	sErrorDescription1 := ' Faulty wiring (Mode sel. swit.  The state of doubled wiring is not matching (Mode sel. switch).';				
	sErrorDescription2 := 'Please check the wiring (Mode sel. switch)';				
					
0047:					
					
	sErrorDescription1 := ' OCL detect.  OCL detect.';				
	sErrorDescription2 := 'Please check the line (O/P Emergency Stop)';				
					
0048:					
					
	sErrorDescription1 := ' Faulty line (Mode Selector SW.  The state of doubled line is not matching (Mode Selector switch).';				
	sErrorDescription2 := 'Please check the line (Mode Selector switch)';				
					
0049:					
					
	sErrorDescription1 := ' Faulty Line (T/B Enable Switc.  The state of doubled line is not matching (T/B Enable Switch).';				
	sErrorDescription2 := 'Please check the line (T/B Enable Switch)';				
					
0050:					
					
	sErrorDescription1 := 'EMG signal is input. (externa.  EMG signal is input. (external).';				
	sErrorDescription2 := 'Check the external emergency stop';				
					
0051:					
					
	sErrorDescription1 := 'EMG line is faulty.(external).  EMG line is faulty.(external).';				
	sErrorDescription2 := 'Check the external emergency stop';				
					
0052:					
					
	sErrorDescription1 := ' EMG signal is input.(Add.Axis.  EMG signal is input.(Add.Axis1).';				
	sErrorDescription2 := 'Check the emergency stop of Additional Axis card';				
					
0053:					
					
	sErrorDescription1 := 'EMG signal is input.(Add.Axis.  EMG signal is input.(Add.Axis).';				
	sErrorDescription2 := 'Check the emergency stop of Additional Axis servo amp.';				
					
0054:					
					
	sErrorDescription1 := ' Faulty wiring (External EMG p.  The state of doubled wiring is not matching (External EMG).';				
	sErrorDescription2 := 'Please check the wiring (External Emergency Stop)';				
					
0060:					
					
	sErrorDescription1 := 'EMG signal is input. (O.Panel.  EMG signal is input. (O.Panel).';				
	sErrorDescription2 := 'Check the O.Panel emergency stop';				
					
0061:					
					
	sErrorDescription1 := 'EMG line is faulty.(0.Panel).  EMG line is faulty.(0.Panel).';				
	sErrorDescription2 := 'Check the O.Panel emergency stop';				
					
0070:					
					
	sErrorDescription1 := 'EMG signal is input. (T.Box).  EMG signal is input. (T.Box).';				
	sErrorDescription2 := 'Check the T.Box emergency stop';				
					
0071:					
					
	sErrorDescription1 := 'EMG line is faulty.(T.Box).  EMG line is faulty.(T.Box).';				
	sErrorDescription2 := 'Check the T.Box emergency stop';				
					
0072:					
					
	sErrorDescription1 := 'EMG cancel operation is fault.  TB cancel switch operation was incorrect.';				
	sErrorDescription2 := 'Check the T/B cancel switch operation';				
					
0073:					
					
	sErrorDescription1 := 'EMG cancel line is faulty.(T..  EMG cancel line is faulty.(T.Box).';				
	sErrorDescription2 := 'Check the EMG cancel line';				
					
0074:					
					
	sErrorDescription1 := 'Faulty line (T/B Enable/Disab.  The state of doubled line is not matching (T/B Enable/Disable).';				
	sErrorDescription2 := 'Please check the line (T/B Enable/Disable)';				
					
0075:					
					
	sErrorDescription1 := 'TB communication error.  Communication between the RC and TB was cut off.';				
	sErrorDescription2 := 'Check TB communication line';				
					
0076:					
					
	sErrorDescription1 := 'TB connection error.  Cannot detect TB connection.';				
	sErrorDescription2 := 'If this error recurs, please contact us';				
					
0077:					
					
	sErrorDescription1 := ' Electric double layer overvol.  A power supply of a substrate in the robot is broken.';				
	sErrorDescription2 := 'Turn the power OFF and contact your service provider';				
					
0079:					
					
	sErrorDescription1 := ' Contactor of converter unit e.  Contactor of converter unit is closed.';				
	sErrorDescription2 := 'Confirm status of contactor of converter unit';				
					
0080:					
					
	sErrorDescription1 := ' Fuse of brake line is blown.  Fuse of brake line is blown.';				
	sErrorDescription2 := 'Change fuse';				
					
0081:					
					
	sErrorDescription1 := ' Fuse is blown.(motor hand I/F.  Fuse is blown.(motor hand I/F).';				
	sErrorDescription2 := 'Change fuse';				
					
0082:					
					
	sErrorDescription1 := 'Fuse is broken (air hand I/F).  Fuse is blown.(air hand I/F).';				
	sErrorDescription2 := 'Change fuse';				
					
0083:					
					
	sErrorDescription1 := 'Fuse is broken(hand input pow.  Fuse is blown.(hand input power).';				
	sErrorDescription2 := 'Change fuse';				
					
0084:					
					
	sErrorDescription1 := 'Fuse is broken(O/P).  Fuse is blown.(O/P).';				
	sErrorDescription2 := 'Change fuse';				
					
0085:					
					
	sErrorDescription1 := ' Fuse is blown.(External EMG).  Open phase in the input power.';				
	sErrorDescription2 := 'Change fuse';				
					
0086:					
					
	sErrorDescription1 := 'Hand module overcurrent.  Hand module is broken.';				
	sErrorDescription2 := 'Change Hand module';				
					
0087:					
					
	sErrorDescription1 := 'Fuse is blown.(Brake).  Fuse is blown.(Brake).';				
	sErrorDescription2 := 'Change fuse';				
					
0088:					
					
	sErrorDescription1 := ' Fuse is blown.(Service I/F).  Fuse is blown.(Service I/F).';				
	sErrorDescription2 := 'Please confirm the input and output current of service I/F. ';				
					
0089:					
					
	sErrorDescription1 := ' Fuse of external battery is b.  Fuse of external battery is blown..';				
	sErrorDescription2 := 'Check that an outside power-supply voltage is 4.5V or less.';				
					
0090:					
					
	sErrorDescription1 := ' Fuse is blown..  Fuse is blown.';				
	sErrorDescription2 := 'Change fuse';				
					
0093:					
					
	sErrorDescription1 := ' Safety relay fuse is blown..  Safety relay fuse is blown..';				
	sErrorDescription2 := 'Change fuse.';				
					
0094:					
					
	sErrorDescription1 := ' The fuse in the T/B was blown.  The fuse in the T/B power supply line was blown..';				
	sErrorDescription2 := 'Please check the earth fault of the T/B cable.';				
					
0097:					
					
	sErrorDescription1 := ' Faulty status (MC).  The state of doubled signal is not matching (MC status).';				
	sErrorDescription2 := 'Turn the power OFF and ON once';				
					
0098:					
					
	sErrorDescription1 := ' Faulty status (SR).  The state of doubled signal is not matching (SR status).';				
	sErrorDescription2 := 'Turn the power OFF and ON once';				
					
0099:					
					
	sErrorDescription1 := ' S/W with an old version is in.  S/W with an old version is installed.';				
	sErrorDescription2 := 'Install the S/W with a correct version';				
					
0100:					
					
	sErrorDescription1 := 'Temperature in the Controlle .  FAN check or Filter at the bottom on Controller becomes old.';				
	sErrorDescription2 := 'Please exchange the filter to new filter or clean up the filter';				
					
0103:					
					
	sErrorDescription1 := ' Temp. in robot CPU is too hig.  Ambient temperature of robot CPU becomes high.';				
	sErrorDescription2 := 'Please lower ambient temperature to the specification range';				
					
0117:					
					
	sErrorDescription1 := ' Power supply error (brake).  The output of the power supply deviated from the specified range.';				
	sErrorDescription2 := 'Turn the power OFF and contact your service provider';				
					
0130:					
					
	sErrorDescription1 := 'System RemoteI/O down.  Communication line of System Remote I/O is illegal.';				
	sErrorDescription2 := 'Check the cable or power supply';				
					
0131:					
					
	sErrorDescription1 := ' Plural Ope-panel are installe.  One operation panel can be installed..';				
	sErrorDescription2 := 'Install only one operation panel.';				
					
0140:					
					
	sErrorDescription1 := 'Fuse is blown.(Safety unit).  Fuse is blown.(Safety unit).';				
	sErrorDescription2 := 'Change fuse';				
					
0141:					
					
	sErrorDescription1 := ' Wiring error of EMGIN connect.  Wiring error of EMGIN connector.';				
	sErrorDescription2 := 'Please confirm the wiring for EMGIN';				
					
0160:					
					
	sErrorDescription1 := 'Cannot use PIO I/F and Unit.  The I/O Channel number of PIO interface and PIO unit overlaps..';				
	sErrorDescription2 := 'Select either of Paralle I/O interface or Paralle I/O unit.';				
					
0162:					
					
	sErrorDescription1 := 'Cannot use PIO I/F and Unit.  The I/O Channel number of PIO interface and PIO unit overlaps..';				
	sErrorDescription2 := 'Select either of Paralle I/O interface or Paralle I/O unit.';				
					
0163:					
					
	sErrorDescription1 := 'Cannot use PIO I/F and Unit.  The I/O Channel number of PIO interface and PIO unit overlaps..';				
	sErrorDescription2 := 'Select either of Paralle I/O interface or Paralle I/O unit.';				
					
0170:					
					
	sErrorDescription1 := 'Parallel I/O interface H/W er.  The card might be broken..';				
	sErrorDescription2 := 'Please exchange the Parallel I/O interface card.';				
					
0172:					
					
	sErrorDescription1 := 'Parallel I/O interface H/W er.  The card might be broken..';				
	sErrorDescription2 := 'Please exchange the Parallel I/O interface card.';				
					
0173:					
					
	sErrorDescription1 := 'Parallel I/O interface H/W er.  The card might be broken..';				
	sErrorDescription2 := 'Please exchange the Parallel I/O interface card.';				
					
0180:					
					
	sErrorDescription1 := 'Fuse is blown.(PIO) （Slot 1-F.  Fuse is blown.(Paralle I/O interface).';				
	sErrorDescription2 := 'Change fuse (Paralle I/O interface)';				
					
0182:					
					
	sErrorDescription1 := 'Fuse is blown.(PIO) （Slot 2-F.  Fuse is blown.(Paralle I/O interface).';				
	sErrorDescription2 := 'Change fuse (Paralle I/O interface)';				
					
0183:					
					
	sErrorDescription1 := 'Fuse is blown.(PIO) （Slot 3-F.  Fuse is blown.(Paralle I/O interface).';				
	sErrorDescription2 := 'Change fuse (Paralle I/O interface)';				
					
0210:					
					
	sErrorDescription1 := ' Power supply error.  The output of the power supply deviated from the specified range.';				
	sErrorDescription2 := 'Turn the power OFF and ON once';				
					
0211:					
					
	sErrorDescription1 := ' Power supply error.  The output of the power supply deviated from the specified range.';				
	sErrorDescription2 := 'Turn the power OFF and ON once';				
					
0212:					
					
	sErrorDescription1 := ' Power supply error.  The output of the power supply deviated from the specified range.';				
	sErrorDescription2 := 'Turn the power OFF and ON once';				
					
0213:					
					
	sErrorDescription1 := ' Power supply error.  The output of the power supply deviated from the specified range.';				
	sErrorDescription2 := 'Turn the power OFF and ON once';				
					
0220:					
					
	sErrorDescription1 := ' Memory error (Main CPU).  Memory error was detected (Main CPU).';				
	sErrorDescription2 := 'Turn the power OFF and ON once';				
					
0230:					
					
	sErrorDescription1 := ' Safety parameter error.  Detect errors in safety parameter value.';				
	sErrorDescription2 := 'Please check the safety parameter setting';				
					
0231:					
					
	sErrorDescription1 := ' Parameter CRC error.  Detect CRC errors in safety parameter.';				
	sErrorDescription2 := 'Please check the safety parameters settings and write parameters';				
					
0241:					
					
	sErrorDescription1 := ' Fault in Safety Communication.  Detect a fault in safety communication.';				
	sErrorDescription2 := 'Turn the power OFF and ON once';				
					
0242:					
					
	sErrorDescription1 := ' Fault in Safety Data.  Detect a fault in safety data.';				
	sErrorDescription2 := 'Turn the power OFF and ON once';				
					
0243:					
					
	sErrorDescription1 := ' Safety function unavailable.  The Safety Function is not supported by this robot.';				
	sErrorDescription2 := 'Disable the safety function';				
					
0260:					
					
	sErrorDescription1 := ' EMG circuit diagnosis error.  Voltage diagnosis error.';				
	sErrorDescription2 := 'Turn the power OFF and ON once';				
					
0270:					
					
	sErrorDescription1 := ' Voltage diagnosis error.  Voltage diagnosis error.';				
	sErrorDescription2 := 'Turn the power OFF and ON once';				
					
0280:					
					
	sErrorDescription1 := ' STO circuit diagnosis error.  STO citcuit error.';				
	sErrorDescription2 := 'Turn the power OFF and ON once';				
					
0290:					
					
	sErrorDescription1 := ' PLD control error.  PLD control error.';				
	sErrorDescription2 := 'Turn the power OFF and ON once';				
					
0300:					
					
	sErrorDescription1 := ' CR800 test H-Error.  General-purpose H-Error for the function test of CR800.';				
	sErrorDescription2 := 'Check the embedded message';				
					
0310:					
					
	sErrorDescription1 := ' Mecha board access error.  Failed in access to a Mecha board.';				
	sErrorDescription2 := 'Please confirm the connection with Mecha board';				
					
0311:					
					
	sErrorDescription1 := ' RemoteI/O unit config error.  The multiple RemoteI/O units which do not support are connected.';				
	sErrorDescription2 := 'Please confirm the constitution of RemoteI/O unit';				
					
0315:					
					
	sErrorDescription1 := ' Can not access the D-device are.  This area cannot be used in duplicate.';				
	sErrorDescription2 := 'Please change the D-device start number in parameter DDEVVLn';				
					
0316:					
					
	sErrorDescription1 := ' The D-device area is out of r.  An area corresponding to the variable type can not be allocated.';				
	sErrorDescription2 := 'Please change the D-device start number in parameter DDEVVLn';				
					
0317:					
					
	sErrorDescription1 := ' The D-device variable duplica.  Cannot be doubly allotted to one variable.';				
	sErrorDescription2 := 'Please change the variable name in parameter DDEVVLn';				
					
0470:					
					
	sErrorDescription1 := ' Abnormality of DB(Add.Axis).  The addition axis dynamic brake is abnormal.';				
	sErrorDescription2 := 'Check the dynamic brake unit and the cable connection';				
					
0490:					
					
	sErrorDescription1 := 'Alarm of fan in the robot.  Fan in the robot might be out of order.';				
	sErrorDescription2 := 'Please exchange the fan in the robot';				
					
0491:					
					
	sErrorDescription1 := 'Alarm of fan1 in the robot.  Fan1 in the robot might be out of order.';				
	sErrorDescription2 := 'Please exchange the fan1 in the robot';				
					
0492:					
					
	sErrorDescription1 := 'Alarm of fan2 in the robot.  Fan2 in the robot might be out of order.';				
	sErrorDescription2 := 'Please exchange the fan2 in the robot';				
					
0493:					
					
	sErrorDescription1 := 'Alarm of fan3 in the robot.  Fan3 in the robot might be out of order.';				
	sErrorDescription2 := 'Please exchange the fan3 in the robot';				
					
0494:					
					
	sErrorDescription1 := 'Alarm of fan4 in the robot.  Fan4 in the robot might be out of order.';				
	sErrorDescription2 := 'Please exchange the fan4 in the robot';				
					
0495:					
					
	sErrorDescription1 := 'Alarm of fan5 in the robot.  Fan5 in the robot might be out of order.';				
	sErrorDescription2 := 'Please exchange the fan5 in the robot';				
					
0496:					
					
	sErrorDescription1 := 'Alarm of fan6 in the robot.  Fan6 in the robot might be out of order.';				
	sErrorDescription2 := 'Please exchange the fan6 in the robot';				
					
0497:					
					
	sErrorDescription1 := 'Alarm of fan7 in the robot.  Fan7 in the robot might be out of order.';				
	sErrorDescription2 := 'Please exchange the fan7 in the robot';				
					
0498:					
					
	sErrorDescription1 := 'Alarm of fan8 in the robot.  Fan8 in the robot might be out of order.';				
	sErrorDescription2 := 'Please exchange the fan8 in the robot';				
					
0500:					
					
	sErrorDescription1 := 'Servo axis setting error.  The setting of the axis number selection switch is illegal.';				
	sErrorDescription2 := 'Confirm the setting of the axis selection switch';				
					
0510:					
					
	sErrorDescription1 := 'The converter setting is ille.  The setting of the external emergency stop mode is illegal.';				
	sErrorDescription2 := 'Correctly set';				
					
0520:					
					
	sErrorDescription1 := 'Robot axis setting illegal.  The axis No is duplicated with another robot axis No.';				
	sErrorDescription2 := 'Correctly set';				
					
0530:					
					
	sErrorDescription1 := 'Servo sys. error (memory).  The servo amplifier memory ICs check sum is illegal.';				
	sErrorDescription2 := 'Turn the power OFF and ON once';				
					
0540:					
					
	sErrorDescription1 := 'Servo sys. error (over run).  The servo amp. / motion task S/W did not end within the specified time.';				
	sErrorDescription2 := 'Turn the power OFF and ON once';				
					
0550:					
					
	sErrorDescription1 := 'Servo sys. error (mag. pole p.  the magnetic pole position signal from encoderis illegal.';				
	sErrorDescription2 := 'Turn the power OFF and ON once';				
					
0560:					
					
	sErrorDescription1 := 'Servo sys. error (A/D）.  the magnetic pole position signal from encoderis illegal.';				
	sErrorDescription2 := 'Turn the power OFF and ON once';				
					
0570:					
					
	sErrorDescription1 := 'Encoder error (EEPROM).  the magnetic pole position signal from encoderis illegal.';				
	sErrorDescription2 := 'Turn the power OFF and ON once';				
					
0580:					
					
	sErrorDescription1 := 'Encoder error (LED).  The LED of encoder has deteriorated.';				
	sErrorDescription2 := 'Turn the power OFF and ON once';				
					
0590:					
					
	sErrorDescription1 := 'Encoder error (position data).  the per rotation position data is illegal.';				
	sErrorDescription2 := 'Turn the power OFF and ON once';				
					
0600:					
					
	sErrorDescription1 := 'Encoder no-signal detection1.  An error was detected in the operation input of the encoder.';				
	sErrorDescription2 := 'Turn the power OFF and ON once';				
					
0610:					
					
	sErrorDescription1 := 'Encoder no-signal detection2.  An error was detected in the operation input of the encoder.';				
	sErrorDescription2 := 'Turn the power OFF and ON once';				
					
0620:					
					
	sErrorDescription1 := 'Servo amplifier LSI error.  An error was detected in the operation of the servo AMP LSI.';				
	sErrorDescription2 := 'Turn the power OFF and ON once';				
					
0630:					
					
	sErrorDescription1 := 'Unused axis servo error.  A power module error occurred in an axis not used.';				
	sErrorDescription2 := 'Turn the power OFF and ON once';				
					
0640:					
					
	sErrorDescription1 := 'System error (ABS CPU).  Error in the CPU of the absolute position linear scale.';				
	sErrorDescription2 := 'Turn the power OFF and ON once';				
					
0650:					
					
	sErrorDescription1 := 'Absolute position error.  Error in the circuit of the absolute position linear scale.';				
	sErrorDescription2 := 'Turn the power OFF and ON once';				
					
0660:					
					
	sErrorDescription1 := 'Incremental position error.  Error in the incremental position detection circuit.';				
	sErrorDescription2 := 'Turn the power OFF and ON once';				
					
0670:					
					
	sErrorDescription1 := 'Encoder CPU error.  An error was detected in the CPU of the encoder.';				
	sErrorDescription2 := 'Turn the power OFF and ON once';				
					
0680:					
					
	sErrorDescription1 := 'Encoder LED error.  Deterioration of the encoder LED was detected.';				
	sErrorDescription2 := 'Turn the power OFF and ON once';				
					
0690:					
					
	sErrorDescription1 := ' regeneration circuit error.  A regenerative transistor or resistor error was detected.';				
	sErrorDescription2 := 'Turn the power OFF and ON once';				
					
0700:					
					
	sErrorDescription1 := 'P.S. external contactor fusin.  The external contactor turned ON even at READY OFF.';				
	sErrorDescription2 := 'Turn the power OFF and ON once';				
					
0710:					
					
	sErrorDescription1 := 'Power supply rush relay error.  The relay on servo cpu card did not turn ON.';				
	sErrorDescription2 := 'Turn the power OFF and ON once';				
					
0711:					
					
	sErrorDescription1 := 'Power supply relay error.  The discharge relay on converter card did not turn ON.';				
	sErrorDescription2 := 'Turn the power OFF and ON once';				
					
0712:					
					
	sErrorDescription1 := ' Converter fuse fusing.  Fuse of a converter fused for a ground fault or short circuit.';				
	sErrorDescription2 := 'Please exchange a fuse of a converter';				
					
0713:					
					
	sErrorDescription1 := ' Encoder power supply fuse tri.  Encoder power supply fuse tripped by ground fault, short circuit.';				
	sErrorDescription2 := 'Turn the power OFF, wait a while, and then turn ON again';				
					
0720:					
					
	sErrorDescription1 := 'Power supply watch dog.  The power supply S/W did not end within the specified time.';				
	sErrorDescription2 := 'Turn the power OFF and ON once';				
					
0730:					
					
	sErrorDescription1 := 'Power supply rush relay fusin.  The rush resistance short-circuit relay did not turn OFF.';				
	sErrorDescription2 := 'Turn the power OFF and ON once';				
					
0740:					
					
	sErrorDescription1 := 'Power supply main circuit err.  The main circuit capacitor was not charged correctly.';				
	sErrorDescription2 := 'Turn the power OFF and ON once';				
					
0742:					
					
	sErrorDescription1 := ' Power supply main circuit err.  A main circuit voltage has decreased because of Safety relay.';				
	sErrorDescription2 := 'Check for errors in the Safety relay';				
					
0743:					
					
	sErrorDescription1 := ' Power supply main circuit err.  A main circuit voltage has decreased because of contactor fail..';				
	sErrorDescription2 := 'Check for errors in the contactor.';				
					
0750:					
					
	sErrorDescription1 := 'Power supply memory error.  An error was detected in the power supply memory circuit.';				
	sErrorDescription2 := 'Turn the power OFF and ON once';				
					
0760:					
					
	sErrorDescription1 := 'Power supply error.  An error was detected in the data comm. with the power supply.';				
	sErrorDescription2 := 'Turn the power OFF and ON once';				
					
0770:					
					
	sErrorDescription1 := 'Power supply process error.  An error occurred in the process cycle of power supply.';				
	sErrorDescription2 := 'Turn the power OFF and ON once';				
					
0780:					
					
	sErrorDescription1 := 'Servo amplifier watch dog.  The Servo amplifier S/W did not end within the specified time.';				
	sErrorDescription2 := 'Turn the power OFF and ON once';				
					
0790:					
					
	sErrorDescription1 := 'Servo amplifier boad error.  An error was detected in the servo amplifier PCB.';				
	sErrorDescription2 := 'Turn the power OFF and ON once';				
					
0800:					
					
	sErrorDescription1 := 'Servo amplifier clock error.  An error was detected in the servo amplifier clock.';				
	sErrorDescription2 := 'Turn the power OFF and ON once';				
					
0810:					
					
	sErrorDescription1 := 'Power supply undervoltage.  Insufficient bus voltage was detected in main circuit.';				
	sErrorDescription2 := 'Check the power supply connection and power supply state';				
					
0820:					
					
	sErrorDescription1 := 'Motor ground fault.  A motor cable ground fault was detected.';				
	sErrorDescription2 := 'Check the motor cables connection and conductivity';				
					
0830:					
					
	sErrorDescription1 := 'Servo amplifier overvoltage.  The main circuit bus voltage exceeded the tolerable value.';				
	sErrorDescription2 := 'Check the power voltage and regenerative resistance value';				
					
0840:					
					
	sErrorDescription1 := 'Instantaneous power failure(S.  The power was OFF for 50msec or more.';				
	sErrorDescription2 := 'Check the power supply connection and power supply state';				
					
0850:					
					
	sErrorDescription1 := 'Power supply voltage incorrec.  Open phase in the input power, or the voltage is outof range.';				
	sErrorDescription2 := 'Check the power supply connection and power supply state';				
					
0860:					
					
	sErrorDescription1 := 'Power supply overvoltage.  The main circuit bus voltage exceeded the tolerable value.';				
	sErrorDescription2 := 'Check the power supply connection and power supply state';				
					
0870:					
					
	sErrorDescription1 := 'Power module overheat (Fan St.  A cooling fan stopped, and overheat occurred.';				
	sErrorDescription2 := 'Check the rotation of fan, and the connector connected to a fan';				
					
0880:					
					
	sErrorDescription1 := 'Power module overheat.  Overheating of the power module (IPM) was detected.';				
	sErrorDescription2 := 'Turn the power OFF, wait a while, and then turn ON again';				
					
0890:					
					
	sErrorDescription1 := 'Servo amplifier motor overhea.  The motor or detectors thermal protector activated.';				
	sErrorDescription2 := 'Turn the power OFF, wait a while, and then turn ON again';				
					
0900:					
					
	sErrorDescription1 := 'Absolute position overspeed.  The absolute position linear scale moved 45mm/s or more.';				
	sErrorDescription2 := 'Turn the power OFF and ON once';				
					
0910:					
					
	sErrorDescription1 := 'Servo amplifier overspeed.  The motor speed rose to 1.2 times the rating.';				
	sErrorDescription2 := 'Turn the power OFF and ON once';				
					
0920:					
					
	sErrorDescription1 := 'Power module overcurrent.  An overcurrent was detected in the  power supply IPM.';				
	sErrorDescription2 := 'Check the motor cables connection and conductivity';				
					
0930:					
					
	sErrorDescription1 := 'Motor overcurrent.  An excessive current flowed to the motor.';				
	sErrorDescription2 := 'Turn the power OFF and ON once';				
					
0940:					
					
	sErrorDescription1 := 'Overload 1.  Run in the overload range set with SVOLL and SVOLT.';				
	sErrorDescription2 := 'Check the load weight and the robot for collisions, etc';				
					
0950:					
					
	sErrorDescription1 := 'Overload 2.  95% or more of max current command continued for 1 sec. or more.';				
	sErrorDescription2 := 'Check the load weight and the robot for collisions, etc';				
					
0960:					
					
	sErrorDescription1 := 'Excessive error 1.  The position error exceeded at servo ON.';				
	sErrorDescription2 := 'Check the load weight and press, etc';				
					
0970:					
					
	sErrorDescription1 := 'Excessive error 2.  The position error exceeded at servo OFF.';				
	sErrorDescription2 := 'Check the moving robot arm by something power';				
					
0980:					
					
	sErrorDescription1 := 'Excessive error 3.  Abnormal motor power line connection.';				
	sErrorDescription2 := 'Check the connection of motor power line';				
					
0990:					
					
	sErrorDescription1 := 'Collision detection 0.  A collision detection method 1 error was detected during the G0.';				
	sErrorDescription2 := 'Release the collision state';				
					
1000:					
					
	sErrorDescription1 := 'Collision detection 1.  A collision detection method 1 error was detected during the G1.';				
	sErrorDescription2 := 'Release the collision state';				
					
1010:					
					
	sErrorDescription1 := 'Collision detection.  Robot collided with something, or COLLVL is too low.';				
	sErrorDescription2 := 'Removal of the factor of a collision, or improve COLLVL';				
					
1020:					
					
	sErrorDescription1 := 'Servo AMP over-regeneration.  Overheating of the regenerative resistor was detected.';				
	sErrorDescription2 := 'Check the regeneration capacity and parameter SVPTYPE';				
					
1030:					
					
	sErrorDescription1 := 'Power supply over-regeneratio.  The power supplys regeneration capacity limit was exceeded.';				
	sErrorDescription2 := 'Wait at least 15min in the power ON state, and then turn OFF';				
					
1040:					
					
	sErrorDescription1 := 'Encoder init communication er.  Initial communication with the encoder was not possible.';				
	sErrorDescription2 := 'Check the encoder cable connection';				
					
1050:					
					
	sErrorDescription1 := ' Encoder init communication er.  Initial communication with the encoder was not possible.';				
	sErrorDescription2 := 'Check the encoder cable connection';				
					
1060:					
					
	sErrorDescription1 := ' Encoder communication error.  Communication between the encoder and detector was cut off.';				
	sErrorDescription2 := 'Check the encoder cable connection';				
					
1070:					
					
	sErrorDescription1 := 'Encoder communication error.  Communication between the encoder and detector was cut off.';				
	sErrorDescription2 := 'Check the encoder cable connection';				
					
1080:					
					
	sErrorDescription1 := 'Servo AMP communication error.  Communication from the RC was cut off.';				
	sErrorDescription2 := 'Check the communication cable connection and conductivity';				
					
1090:					
					
	sErrorDescription1 := 'Servo AMP initialization erro.  Initialization of the servo amplifier failed.';				
	sErrorDescription2 := 'Check the servo axis settings (parameters, rotary switches)';				
					
1100:					
					
	sErrorDescription1 := 'Servo com. receive error.  Abnormality occurred in data reception from a servo amplifier.';				
	sErrorDescription2 := 'Check the communication cable connection and conductivity';				
					
1110:					
					
	sErrorDescription1 := 'Servo com. receive error.  Abnormality occurred in data reception from a servo amplifier.';				
	sErrorDescription2 := 'Check the communication cable connection and conductivity';				
					
1120:					
					
	sErrorDescription1 := 'Encoder ABS position data los.  The absolute position data in the detector was lost.';				
	sErrorDescription2 := 'Check the battery voltage and detector cable';				
					
1130:					
					
	sErrorDescription1 := 'Encoder per rotation data err.  An error was detected in the encoders per rotation data.';				
	sErrorDescription2 := 'Check the repeatability and ambient environment';				
					
1140:					
					
	sErrorDescription1 := 'SRV-AMP Comm. data error (CRC.  A CRC error was detected in the data from the RC.';				
	sErrorDescription2 := 'Check the communication cable connection and conductivity';				
					
1150:					
					
	sErrorDescription1 := 'Large command position.  The command position from the RC is abnormally large.';				
	sErrorDescription2 := 'Check the communication cable connection and conductivity';				
					
1160:					
					
	sErrorDescription1 := 'SRV-AMP Comm. error (frame).  An error was detected in the communication frame from the RC.';				
	sErrorDescription2 := 'Check the communication cable connection and conductivity';				
					
1170:					
					
	sErrorDescription1 := 'SRV-AMP Comm. error (info).  Error in the communication information from the RC.';				
	sErrorDescription2 := 'Check the communication cable connection and conductivity';				
					
1180:					
					
	sErrorDescription1 := 'Servo amplifier feedback erro.  A pulse was skipped in the detector feedback signal.';				
	sErrorDescription2 := 'Check the encoder cable connection and conductivity';				
					
1190:					
					
	sErrorDescription1 := 'Servo amplifier feedback erro.  A deviation occurred in the motor end and machine end positions.';				
	sErrorDescription2 := 'Check the encoder';				
					
1200:					
					
	sErrorDescription1 := 'SRV-AMP Comm. data error (CRC.  CRC error in the communication data from the servo amplifier.';				
	sErrorDescription2 := 'Check the communication cable connection and conductivity';				
					
1210:					
					
	sErrorDescription1 := 'SRV-AMP Comm. data error (ID).  Data ID error in the communication data from the servo AMP.';				
	sErrorDescription2 := 'Check the communication cable connection and conductivity';				
					
1220:					
					
	sErrorDescription1 := 'SRV-AMP Comm. data error(axis.  Axis No error in the communication data from the servo AMP.';				
	sErrorDescription2 := 'Check the communication cable connection and conductivity';				
					
1230:					
					
	sErrorDescription1 := 'SRV-AMP Comm. data error(SubI.  Sub ID error in the communication data from the servo AMP.';				
	sErrorDescription2 := 'Check the communication cable connection and conductivity';				
					
1240:					
					
	sErrorDescription1 := 'SRV-AMP Comm. data error(fram.  No. of frames error in the communication data from servo AMP.';				
	sErrorDescription2 := 'Check the communication cable connection and conductivity';				
					
1250:					
					
	sErrorDescription1 := 'Servo amplifier parameter err.  An error was detected in the servo parameter.';				
	sErrorDescription2 := 'Change the servo parameter to an appropriate value';				
					
1360:					
					
	sErrorDescription1 := ' Absolute position counter err.  The counter of absolute position is illegal.';				
	sErrorDescription2 := 'Check the repeatability and ambient environment';				
					
1380:					
					
	sErrorDescription1 := ' Removing control axis (servo).  The axis removable command has been input from the controller.';				
	sErrorDescription2 := 'Reset the axis removable command';				
					
1390:					
					
	sErrorDescription1 := 'Emergency stop (Servo amplifi.  The emergency stop command has been input from the RC.';				
	sErrorDescription2 := 'Release the emergency stop state';				
					
1410:					
					
	sErrorDescription1 := 'Instantaneous power failure(S.  The power was momentarily interrupted.';				
	sErrorDescription2 := 'Check power spec., and wiring of power and external EMG. stop';				
					
1440:					
					
	sErrorDescription1 := 'System error (servo 1).  Trouble occurred in the current processing CPU.';				
	sErrorDescription2 := 'Turn the power OFF and ON';				
					
1450:					
					
	sErrorDescription1 := 'Instantaneous power interrupt.  The power was momentarily interrupted at the power supply.';				
	sErrorDescription2 := 'Check power spec., and wiring of power and external EMG. stop';				
					
1460:					
					
	sErrorDescription1 := 'Power supply overcurrent.  Overcurrent in the power module in the power supply.';				
	sErrorDescription2 := 'Check the AC power line, or change the power supply';				
					
1470:					
					
	sErrorDescription1 := 'Frequency error.  AC frequency is out of range.';				
	sErrorDescription2 := 'Check the AC power line frequency, or change the power supply';				
					
1480:					
					
	sErrorDescription1 := 'Power supply parameter error.  Illegal at the power supply parameter.';				
	sErrorDescription2 := 'Set the correct parameter';				
					
1490:					
					
	sErrorDescription1 := 'Power supply overheat.  Overheating of the power module or regenerative resistance.';				
	sErrorDescription2 := 'Check the fan on rear of power supply';				
					
1491:					
					
	sErrorDescription1 := ' Illegal converter thermal  se.  Overheating of  servo AMP converter..';				
	sErrorDescription2 := 'Turn the power OFF, wait a while, and then turn ON again.';				
					
1492:					
					
	sErrorDescription1 := ' Power supply converter overhe.  Overheating of the converter was detected.';				
	sErrorDescription2 := 'Turn the power OFF, wait a while, and then turn ON again';				
					
1493:					
					
	sErrorDescription1 := ' Rush resistance overheat.  Overheating of the rush resistance was detected.';				
	sErrorDescription2 := 'Turn the power OFF, wait a while, and then turn ON again';				
					
1494:					
					
	sErrorDescription1 := ' Discharge resistance overheat.  Overheating of the discharge resistance was detected.';				
	sErrorDescription2 := 'Turn the power OFF, wait a while, and then turn ON again';				
					
1500:					
					
	sErrorDescription1 := 'Motor combination error.  Illegal combination with additional servo amp and motor.';				
	sErrorDescription2 := 'Use additional servo amp with correctly combination';				
					
1510:					
					
	sErrorDescription1 := 'SRV-AMP USB comm. Error.  A communication error was detected between the servo amp and PC.';				
	sErrorDescription2 := 'Check the communication cable connection and conductivity';				
					
1530:					
					
	sErrorDescription1 := ' Encoder memory error.  .';				
	sErrorDescription2 := '';				
					
1540:					
					
	sErrorDescription1 := 'Communication error between u.  The transmission data between servo amplifier units is illegal.';				
	sErrorDescription2 := 'Check the communication cable connection and conductivity';				
					
1550:					
					
	sErrorDescription1 := 'Emergency stop is a breakdown.  The external emergency stop input is illegal.';				
	sErrorDescription2 := 'Turn the power OFF and ON once';				
					
1561:					
					
	sErrorDescription1 := 'Excessive error 4.  Axis moved during servo on process.';				
	sErrorDescription2 := 'It is necessary to change some parts when not improvement';				
					
1570:					
					
	sErrorDescription1 := 'Non-registered servo error.  A non-registered servo error occurred.';				
	sErrorDescription2 := 'If the warning cannot be reset, turn the power OFF and ON';				
					
1590:					
					
	sErrorDescription1 := ' System error (illegal EMG).  An non-registered emergency stop was input.';				
	sErrorDescription2 := '';				
					
1600:					
					
	sErrorDescription1 := 'System error (No robot setted.  None of the robots are set.';				
	sErrorDescription2 := 'Set the robots for at least one unit';				
					
1601:					
					
	sErrorDescription1 := ' Unmatched robot model.  Robot arm that connection is not correct.';				
	sErrorDescription2 := 'Please confirm the connected robot arm';				
					
1610:					
					
	sErrorDescription1 := 'System error (illegal MEMECH).  The setting parameter MEMECH is illegal.';				
	sErrorDescription2 := 'Set the correct MEMECH';				
					
1680:					
					
	sErrorDescription1 := 'Cannot servo ON (timeout).  The servo did not turn ON within the specified time.';				
	sErrorDescription2 := 'Check for errors in the servo amplifier';				
					
1681:					
					
	sErrorDescription1 := 'Unexpected servo OFF.  The servo turned OFF unexpectedly.';				
	sErrorDescription2 := 'Check for errors in the servo amplifier';				
					
1682:					
					
	sErrorDescription1 := ' Servo ON Timeout(Safety relay.  A main circuit voltage did not rise because of Safety relay.';				
	sErrorDescription2 := 'Check for errors in the Safety relay';				
					
1683:					
					
	sErrorDescription1 := ' Servo ON Timeout.(Contactor).  A main circuit voltage did not rise because of contactor welded..';				
	sErrorDescription2 := 'Check for errors in the contactor.';				
					
1790:					
					
	sErrorDescription1 := 'Illegal parameter (MEJAR).  The setting of parameter MEJAR is illegal.';				
	sErrorDescription2 := 'Correct the parameter MEJAR';				
					
1800:					
					
	sErrorDescription1 := 'Illegal parameter (MEMAR).  The setting of parameter MEMAR is illegal.';				
	sErrorDescription2 := 'Correct the parameter MEMAR';				
					
1810:					
					
	sErrorDescription1 := 'Illegal parameter (USERORG).  The setting of parameter USERORG is illegal.';				
	sErrorDescription2 := 'Correct the parameter USERORG';				
					
1861:					
					
	sErrorDescription1 := 'Illegal parameter (J1OFFSET).  The setting of parameter J1OFFSET is illegal.';				
	sErrorDescription2 := 'Correct the 2nd element of parameter J1OFFSET';				
					
1881:					
					
	sErrorDescription1 := 'Cooling fan stopped (add. axi.  Cooling fan of the add. axis amp. J1 might be out of order.';				
	sErrorDescription2 := 'Please exchange the cooling fan';				
					
1882:					
					
	sErrorDescription1 := 'Cooling fan stopped (add. axi.  Cooling fan of the add. axis amp. J2 might be out of order.';				
	sErrorDescription2 := 'Please exchange the cooling fan';				
					
1883:					
					
	sErrorDescription1 := 'Cooling fan stopped (add. axi.  Cooling fan of the add. axis amp. J3 might be out of order.';				
	sErrorDescription2 := 'Please exchange the cooling fan';				
					
1884:					
					
	sErrorDescription1 := 'Cooling fan stopped (add. axi.  Cooling fan of the add. axis amp. J4 might be out of order.';				
	sErrorDescription2 := 'Please exchange the cooling fan';				
					
1885:					
					
	sErrorDescription1 := 'Cooling fan stopped (add. axi.  Cooling fan of the add. axis amp. J5 might be out of order.';				
	sErrorDescription2 := 'Please exchange the cooling fan';				
					
1886:					
					
	sErrorDescription1 := 'Cooling fan stopped (add. axi.  Cooling fan of the add. axis amp. J6 might be out of order.';				
	sErrorDescription2 := 'Please exchange the cooling fan';				
					
1887:					
					
	sErrorDescription1 := 'Cooling fan stopped (add. axi.  Cooling fan of the add. axis amp. J7 might be out of order.';				
	sErrorDescription2 := 'Please exchange the cooling fan';				
					
1888:					
					
	sErrorDescription1 := 'Cooling fan stopped (add. axi.  Cooling fan of the add. axis amp. J8 might be out of order.';				
	sErrorDescription2 := 'Please exchange the cooling fan';				
					
1900:					
					
	sErrorDescription1 := 'Cooling fan stopped (pow. sup.  The power supply cooling fan stopped.';				
	sErrorDescription2 := 'Confirm the rotation of the power supply cooling fan';				
					
1950:					
					
	sErrorDescription1 := ' Additional axis AMP error.  Alarm of the additional axis servo amplifier was detected.';				
	sErrorDescription2 := 'Please refer to the manual of servo amplifier.';				
					
2031:					
					
	sErrorDescription1 := 'Illegal parameter(JOGTSJ,JOGJ.  Illegal parameter(JOGTSJ,JOGJSP).';				
	sErrorDescription2 := 'Set value under 5';				
					
2090:					
					
	sErrorDescription1 := 'In interference zone n.  Movement inside the user-defined area range was attempted.';				
	sErrorDescription2 := 'Adjust the position data';				
					
2111:					
					
	sErrorDescription1 := 'Free plane 1 overrun.  Movement outside the free plane 1 was attempted.';				
	sErrorDescription2 := 'Change the position data';				
					
2112:					
					
	sErrorDescription1 := 'Free plane 2 overrun.  Movement outside the free plane 2 was attempted.';				
	sErrorDescription2 := 'Change the position data';				
					
2113:					
					
	sErrorDescription1 := 'Free plane 3 overrun.  Movement outside the free plane 3 was attempted.';				
	sErrorDescription2 := 'Change the position data';				
					
2114:					
					
	sErrorDescription1 := 'Free plane 4 overrun.  Movement outside the free plane 4 was attempted.';				
	sErrorDescription2 := 'Change the position data';				
					
2115:					
					
	sErrorDescription1 := 'Free plane 5 overrun.  Movement outside the free plane 5 was attempted.';				
	sErrorDescription2 := 'Change the position data';				
					
2116:					
					
	sErrorDescription1 := 'Free plane 6 overrun.  Movement outside the free plane 6 was attempted.';				
	sErrorDescription2 := 'Change the position data';				
					
2117:					
					
	sErrorDescription1 := 'Free plane 7 overrun.  Movement outside the free plane 7 was attempted.';				
	sErrorDescription2 := 'Change the position data';				
					
2118:					
					
	sErrorDescription1 := 'Free plane 8 overrun.  Movement outside the free plane 8 was attempted.';				
	sErrorDescription2 := 'Change the position data';				
					
2119:					
					
	sErrorDescription1 := ' Free plane 9 overrun.  Movement outside the free plane 9 was attempted.';				
	sErrorDescription2 := 'Change the position data';				
					
2120:					
					
	sErrorDescription1 := ' Free plane 10 overrun.  Movement outside the free plane 10 was attempted.';				
	sErrorDescription2 := 'Change the position data';				
					
2121:					
					
	sErrorDescription1 := ' Free plane 11 overrun.  Movement outside the free plane 11 was attempted.';				
	sErrorDescription2 := 'Change the position data';				
					
2122:					
					
	sErrorDescription1 := ' Free plane 12 overrun.  Movement outside the free plane 12 was attempted.';				
	sErrorDescription2 := 'Change the position data';				
					
2123:					
					
	sErrorDescription1 := ' Free plane 13 overrun.  Movement outside the free plane 13 was attempted.';				
	sErrorDescription2 := 'Change the position data';				
					
2124:					
					
	sErrorDescription1 := ' Free plane 14 overrun.  Movement outside the free plane 14 was attempted.';				
	sErrorDescription2 := 'Change the position data';				
					
2125:					
					
	sErrorDescription1 := ' Free plane 15 overrun.  Movement outside the free plane 15 was attempted.';				
	sErrorDescription2 := 'Change the position data';				
					
2126:					
					
	sErrorDescription1 := ' Free plane 16 overrun.  Movement outside the free plane 16 was attempted.';				
	sErrorDescription2 := 'Change the position data';				
					
2129:					
					
	sErrorDescription1 := 'Free plane limit data illegal.  The free plane data setting value is illegal.';				
	sErrorDescription2 := 'Set the correct free plane setting data';				
					
2130:					
					
	sErrorDescription1 := 'Speed is excessive (command).  The axis speed limit was exceeded.';				
	sErrorDescription2 := 'Reduce the robot motion speed,insert an OVRD,ACCEL or SPD';				
					
2131:					
					
	sErrorDescription1 := 'J1 Speed is excessive (comman.  The axis J1 speed limit was exceeded.';				
	sErrorDescription2 := 'Reduce the robot motion speed,insert an OVRD,ACCEL or SPD';				
					
2132:					
					
	sErrorDescription1 := 'J2 Speed is excessive (comman.  The axis J2 speed limit was exceeded.';				
	sErrorDescription2 := 'Reduce the robot motion speed,insert an OVRD,ACCEL or SPD';				
					
2133:					
					
	sErrorDescription1 := 'J3 Speed is excessive (comman.  The axis J3 speed limit was exceeded.';				
	sErrorDescription2 := 'Reduce the robot motion speed,insert an OVRD,ACCEL or SPD';				
					
2134:					
					
	sErrorDescription1 := 'J4 Speed is excessive (comman.  The axis J4 speed limit was exceeded.';				
	sErrorDescription2 := 'Reduce the robot motion speed,insert an OVRD,ACCEL or SPD';				
					
2135:					
					
	sErrorDescription1 := 'J5 Speed is excessive (comman.  The axis J5 speed limit was exceeded.';				
	sErrorDescription2 := 'Reduce the robot motion speed,insert an OVRD,ACCEL or SPD';				
					
2136:					
					
	sErrorDescription1 := 'J6 Speed is excessive (comman.  The axis J6 speed limit was exceeded.';				
	sErrorDescription2 := 'Reduce the robot motion speed,insert an OVRD,ACCEL or SPD';				
					
2137:					
					
	sErrorDescription1 := 'J7 Speed is excessive (comman.  The axis J7 speed limit was exceeded.';				
	sErrorDescription2 := 'Reduce the robot motion speed,insert an OVRD,ACCEL or SPD';				
					
2138:					
					
	sErrorDescription1 := 'J8 Speed is excessive (comman.  The axis J8 speed limit was exceeded.';				
	sErrorDescription2 := 'Reduce the robot motion speed,insert an OVRD,ACCEL or SPD';				
					
2140:					
					
	sErrorDescription1 := 'ABS limit over.  ABS limit over.';				
	sErrorDescription2 := 'JOG operation with LS release operation';				
					
2141:					
					
	sErrorDescription1 := 'J1 +ABS limit over.  J1 +ABS limit over.';				
	sErrorDescription2 := 'JOG operation with LS release operation';				
					
2142:					
					
	sErrorDescription1 := 'J2 +ABS limit over.  J2 +ABS limit over.';				
	sErrorDescription2 := 'JOG operation with LS release operation';				
					
2143:					
					
	sErrorDescription1 := 'J3 +ABS limit over.  J3 +ABS limit over.';				
	sErrorDescription2 := 'JOG operation with LS release operation';				
					
2144:					
					
	sErrorDescription1 := 'J4 +ABS limit over.  J4 +ABS limit over.';				
	sErrorDescription2 := 'JOG operation with LS release operation';				
					
2145:					
					
	sErrorDescription1 := 'J5 +ABS limit over.  J5 +ABS limit over.';				
	sErrorDescription2 := 'JOG operation with LS release operation';				
					
2146:					
					
	sErrorDescription1 := 'J6 +ABS limit over.  J6 +ABS limit over.';				
	sErrorDescription2 := 'JOG operation with LS release operation';				
					
2147:					
					
	sErrorDescription1 := 'J7 +ABS limit over.  J7 +ABS limit over.';				
	sErrorDescription2 := 'JOG operation with LS release operation';				
					
2148:					
					
	sErrorDescription1 := 'J8 +ABS limit over.  J8 +ABS limit over.';				
	sErrorDescription2 := 'JOG operation with LS release operation';				
					
2151:					
					
	sErrorDescription1 := 'J1 -ABS limit over.  J1 -ABS limit over.';				
	sErrorDescription2 := 'JOG operation with LS release operation';				
					
2152:					
					
	sErrorDescription1 := 'J2 -ABS limit over.  J2 -ABS limit over.';				
	sErrorDescription2 := 'JOG operation with LS release operation';				
					
2153:					
					
	sErrorDescription1 := 'J3 -ABS limit over.  J3 -ABS limit over.';				
	sErrorDescription2 := 'JOG operation with LS release operation';				
					
2154:					
					
	sErrorDescription1 := 'J4 -ABS limit over.  J4 -ABS limit over.';				
	sErrorDescription2 := 'JOG operation with LS release operation';				
					
2155:					
					
	sErrorDescription1 := 'J5 -ABS limit over.  J5 -ABS limit over.';				
	sErrorDescription2 := 'JOG operation with LS release operation';				
					
2156:					
					
	sErrorDescription1 := 'J6 -ABS limit over.  J6 -ABS limit over.';				
	sErrorDescription2 := 'JOG operation with LS release operation';				
					
2157:					
					
	sErrorDescription1 := 'J7 -ABS limit over.  J7 -ABS limit over.';				
	sErrorDescription2 := 'JOG operation with LS release operation';				
					
2158:					
					
	sErrorDescription1 := 'J8 -ABS limit over.  J8 -ABS limit over.';				
	sErrorDescription2 := 'JOG operation with LS release operation';				
					
2160:					
					
	sErrorDescription1 := 'Joint angle exceeds the limit.  Joint angle exceeds the limit.';				
	sErrorDescription2 := 'Change the position data';				
					
2161:					
					
	sErrorDescription1 := 'J1 (+) angle exceeds the limi.  J1(+) angle exceeds the limit.';				
	sErrorDescription2 := 'Change the position data';				
					
2162:					
					
	sErrorDescription1 := 'J2 (+) angle exceeds the limi.  J2(+) angle exceeds the limit.';				
	sErrorDescription2 := 'Change the position data';				
					
2163:					
					
	sErrorDescription1 := 'J3 (+) angle exceeds the limi.  J3(+) angle exceeds the limit.';				
	sErrorDescription2 := 'Change the position data';				
					
2164:					
					
	sErrorDescription1 := 'J4 (+) angle exceeds the limi.  J4(+) angle exceeds the limit.';				
	sErrorDescription2 := 'Change the position data';				
					
2165:					
					
	sErrorDescription1 := 'J5 (+) angle exceeds the limi.  J5(+) angle exceeds the limit.';				
	sErrorDescription2 := 'Change the position data';				
					
2166:					
					
	sErrorDescription1 := 'J6 (+) angle exceeds the limi.  J6(+) angle exceeds the limit.';				
	sErrorDescription2 := 'Change the position data';				
					
2167:					
					
	sErrorDescription1 := 'J7 (+) angle exceeds the limi.  J7(+) angle exceeds the limit.';				
	sErrorDescription2 := 'Change the position data';				
					
2168:					
					
	sErrorDescription1 := 'J8 (+) angle exceeds the limi.  J8(+) angle exceeds the limit.';				
	sErrorDescription2 := 'Change the position data';				
					
2171:					
					
	sErrorDescription1 := 'J1 (-) angle exceeds the limi.  J1(-) angle exceeds the limit.';				
	sErrorDescription2 := 'Change the position data';				
					
2172:					
					
	sErrorDescription1 := 'J2 (-) angle exceeds the limi.  J2(-) angle exceeds the limit.';				
	sErrorDescription2 := 'Change the position data';				
					
2173:					
					
	sErrorDescription1 := 'J3 (-) angle exceeds the limi.  J3(-) angle exceeds the limit.';				
	sErrorDescription2 := 'Change the position data';				
					
2174:					
					
	sErrorDescription1 := 'J4 (-) angle exceeds the limi.  J4(-) angle exceeds the limit.';				
	sErrorDescription2 := 'Change the position data';				
					
2175:					
					
	sErrorDescription1 := 'J5 (-) angle exceeds the limi.  J5(-) angle exceeds the limit.';				
	sErrorDescription2 := 'Change the position data';				
					
2176:					
					
	sErrorDescription1 := 'J6 (-) angle exceeds the limi.  J6(-) angle exceeds the limit.';				
	sErrorDescription2 := 'Change the position data';				
					
2177:					
					
	sErrorDescription1 := 'J7 (-) angle exceeds the limi.  J7(-) angle exceeds the limit.';				
	sErrorDescription2 := 'Change the position data';				
					
2178:					
					
	sErrorDescription1 := 'J8 (-) angle exceeds the limi.  J8(-) angle exceeds the limit.';				
	sErrorDescription2 := 'Change the position data';				
					
2180:					
					
	sErrorDescription1 := 'X,Y,Z data exceeds the limit.  X,Y,Z data exceeds the limit.';				
	sErrorDescription2 := 'Change the position data';				
					
2181:					
					
	sErrorDescription1 := 'X(+) data exceeds the limit.  X(+) data exceeds the limit.';				
	sErrorDescription2 := 'Change the position data';				
					
2182:					
					
	sErrorDescription1 := 'Y(+) data exceeds the limit.  Y(+) data exceeds the limit.';				
	sErrorDescription2 := 'Change the position data';				
					
2183:					
					
	sErrorDescription1 := 'Z(+) data exceeds the limit.  Z(+) data exceeds the limit.';				
	sErrorDescription2 := 'Change the position data';				
					
2191:					
					
	sErrorDescription1 := 'X(-) data exceeds the limit.  X(-) data exceeds the limit.';				
	sErrorDescription2 := 'Change the position data';				
					
2192:					
					
	sErrorDescription1 := 'Y(-) data exceeds the limit.  Y(-) data exceeds the limit.';				
	sErrorDescription2 := 'Change the position data';				
					
2193:					
					
	sErrorDescription1 := 'Z(-) data exceeds the limit.  Z(-) data exceeds the limit.';				
	sErrorDescription2 := 'Change the position data';				
					
2200:					
					
	sErrorDescription1 := ' SLP (ROBOT position error).  Safety Position monitoring detected over the position limits.';				
	sErrorDescription2 := 'Please confirm the robot movement or related parameter setting';				
					
2210:					
					
	sErrorDescription1 := ' STR (ROBOT torque error).  Safety Torque Range monitoring detected over the torque thresh..';				
	sErrorDescription2 := 'Please confirm the robot movement or related parameter setting';				
					
2220:					
					
	sErrorDescription1 := ' Mismatch of Dual Safety Input.  State of the redundant wiring do not match (Dual Safty Input).';				
	sErrorDescription2 := 'Please check the wiring or parameter';				
					
2230:					
					
	sErrorDescription1 := ' Mismatch of Dual Safety Outpu.  State of the redundant wiring do not match (Dual Safty Output).';				
	sErrorDescription2 := 'If this error recurs, please contact us';				
					
2231:					
					
	sErrorDescription1 := ' Mismatch of Dual Safety Outpu.  State of Dual Safty Output and the feedback do not match.';				
	sErrorDescription2 := 'If this error recurs, please contact us';				
					
2240:					
					
	sErrorDescription1 := ' Origin data was changed.  Origin data was changed under the position monitor processing.';				
	sErrorDescription2 := 'Turn the power OFF and ON once';				
					
2260:					
					
	sErrorDescription1 := ' Safety function is not execut.  Extended safety unit of the robot safety option is not installed.';				
	sErrorDescription2 := 'Please install the extended safety unit';				
					
2261:					
					
	sErrorDescription1 := ' Extended safety units No. er.  The extended safety unit’s station No. is illegal.';				
	sErrorDescription2 := 'Set the extended safety unit’s station No. to 2';				
					
2280:					
					
	sErrorDescription1 := ' SS1 deceleration time exceede.  The robot did not stop within deceleration time from SS1 enabled.';				
	sErrorDescription2 := 'Please confirm the robot movement or related parameter setting';				
					
2281:					
					
	sErrorDescription1 := ' SS2 deceleration time exceede.  The robot did not stop within deceleration time from SS2 enabled.';				
	sErrorDescription2 := 'Please confirm the robot movement or related parameter setting';				
					
2282:					
					
	sErrorDescription1 := ' SOS error.  Detect the change of position FB on SOS.';				
	sErrorDescription2 := 'Please check external force or related parameter settings';				
					
2300:					
					
	sErrorDescription1 := ' SLS (Joint Speed Error).  Speed monitor detected the speed over.';				
	sErrorDescription2 := 'Please confirm the robot movement or related parameter setting';				
					
2310:					
					
	sErrorDescription1 := ' SLS (XYZ Speed Error).  Speed monitor detected the speed over.';				
	sErrorDescription2 := 'Please confirm the robot movement or related parameter setting';				
					
2320:					
					
	sErrorDescription1 := ' SF (Robot control error).  Command position and F/B position are not corresponding.';				
	sErrorDescription2 := 'Please confirm the robot movement and presence of interference';				
					
2330:					
					
	sErrorDescription1 := ' SF (Servo control error).  Abnormality of Servo Control was detected.';				
	sErrorDescription2 := 'Please confirm the robot movement and presence of interference';				
					
2340:					
					
	sErrorDescription1 := ' SF (Motion command error).  Abnormality of Command Position was detected.';				
	sErrorDescription2 := 'Turn the power OFF and ON once';				
					
2350:					
					
	sErrorDescription1 := ' SLS (Motor drive command erro.  Speed monitor (Servo) detected the position command speed excess.';				
	sErrorDescription2 := 'Turn the power OFF and ON once';				
					
2360:					
					
	sErrorDescription1 := ' SF (Encoder data error).  Abnormality of Encoder Data was detected.';				
	sErrorDescription2 := 'Turn the power OFF and ON once';				
					
2370:					
					
	sErrorDescription1 := ' SF (Process error).  The Safety Function is not normally executed.';				
	sErrorDescription2 := 'Turn the power OFF and ON once';				
					
2380:					
					
	sErrorDescription1 := ' SF (SCPU Process error).  Abnormality of the Safety Function was detected.';				
	sErrorDescription2 := 'Turn the power OFF and ON once';				
					
2420:					
					
	sErrorDescription1 := ' Collision avoidance comm. err.  Collision avoidance comm. error.';				
	sErrorDescription2 := 'Check the robot controller';				
					
2500:					
					
	sErrorDescription1 := 'Tracking encoder data error.  An error was detected in the tracking encoder data.';				
	sErrorDescription2 := 'Check the repeatability and ambient environment';				
					
2570:					
					
	sErrorDescription1 := ' Installation slot error..  Q173DPX is installed in slot 0-2 of a basic base..';				
	sErrorDescription2 := 'Install Q173DPX to slot 3-11.';				
					
2630:					
					
	sErrorDescription1 := ' Setting the value of DISPCTYP.  Out of range value is set to DISPCTYP.';				
	sErrorDescription2 := 'Please confirm the value of DISPCTYP';				
					
2640:					
					
	sErrorDescription1 := ' Add axis FLS signal is input.  Add axis FLS signal is input.';				
	sErrorDescription2 := 'JOG operation with LS release operation';				
					
2650:					
					
	sErrorDescription1 := ' Add axis RLS signal is input.  Add axis RLS signal is input.';				
	sErrorDescription2 := 'JOG operation with LS release operation';				
					
2663:					
					
	sErrorDescription1 := ' Origin data was changed.  Origin data was changed about the base cooperation target axis.';				
	sErrorDescription2 := 'Turn the power OFF and ON once';				
					
2760:					
					
	sErrorDescription1 := ' Correction limit (F.Ctrl).  The correction value of the force control exceeded the limit.';				
	sErrorDescription2 := 'Please confirm the movement of the robot';				
					
2770:					
					
	sErrorDescription1 := ' exceeds the joint limit.  Position of force control exceeds the joint limit.';				
	sErrorDescription2 := 'Please revice the position';				
					
2780:					
					
	sErrorDescription1 := ' exceeds the speed limit.  Position of force control exceeds the speed limit.';				
	sErrorDescription2 := 'Please revice the operation';				
					
2820:					
					
	sErrorDescription1 := 'Illegal ACCEL ratio.  Illegal ACCEL ratio.';				
	sErrorDescription2 := 'Set the correct ACCEL ratio';				
					
2840:					
					
	sErrorDescription1 := 'System error (ipol parameters.  Parameters setting is illegal.';				
	sErrorDescription2 := 'Set the correct parameters';				
					
2850:					
					
	sErrorDescription1 := 'System error (ipol norm).  System error (ipol norm).';				
	sErrorDescription2 := 'Please call S.C.';				
					
2860:					
					
	sErrorDescription1 := 'System error (ipol type).  Illegal interpolation type.';				
	sErrorDescription2 := 'Please call S.C.';				
					
2870:					
					
	sErrorDescription1 := 'System error(ipol data undef).  Ipol data is undefined.';				
	sErrorDescription2 := 'Please call S.C.';				
					
2880:					
					
	sErrorDescription1 := 'System error (ipol data area).  No more ipol data area.';				
	sErrorDescription2 := 'Please call S.C.';				
					
2890:					
					
	sErrorDescription1 := 'System error (undefined err).  System error (undefined err).';				
	sErrorDescription2 := 'Please call S.C.';				
					
3983:					
					
	sErrorDescription1 := 'Cannot execute CNT movement.  A structural flag or the angle of the joint is not corresponding.';				
	sErrorDescription2 := 'It surely positions it by DLY command etc';				
					
3985:					
					
	sErrorDescription1 := 'Cannot be passsed (singularit.  Robot passes position which is very near the singular point.';				
	sErrorDescription2 := 'Adjust the teaching position';				
					
3988:					
					
	sErrorDescription1 := ' Cannot calculate the position.  Position of force control could not convert a joint angle.';				
	sErrorDescription2 := 'Please revice the position';				
					
5000:					
					
	sErrorDescription1 := 'TB Enable key is ON.  The TB Enable key was ON in the AUTO mode.';				
	sErrorDescription2 := 'OFF the TB Enable key, or enter the TEACH mode';				
					
6000:					
					
	sErrorDescription1 := ' Please execute the all backup.  New error log information was made..';				
	sErrorDescription2 := 'You can reset the error,if "SPCERR" input is ON (Rising edge).';				
					
6100:					
					
	sErrorDescription1 := ' The module is not installed.  The module for the Network Base card is not installed.';				
	sErrorDescription2 := 'Please install the module for the Network Base card';				
					
6101:					
					
	sErrorDescription1 := ' Unsupported module is install.  Unsupported module is installed in the Network Base card.';				
	sErrorDescription2 := 'Please exchange the module';				
					
6110:					
					
	sErrorDescription1 := ' More TZ535 cards are installe.  Only one TZ535 card can be installed.';				
	sErrorDescription2 := 'Please install only one TZ535 card';				
					
6111:					
					
	sErrorDescription1 := ' Other field cards are install.  Only one fieldbus card can be installed.';				
	sErrorDescription2 := 'Only one fieldbus card is installed';				
					
6120:					
					
	sErrorDescription1 := ' Network Base card failure.  Abnormality of the Network Base card is detected.';				
	sErrorDescription2 := 'Please exchange the Network Base card';				
					
6140:					
					
	sErrorDescription1 := ' Parameter error.  Parameter setting is illegal.';				
	sErrorDescription2 := 'Please check the parameter setting';				
					
6510:					
					
	sErrorDescription1 := 'RS232C Parameter illgal.  Setup the parameter.';				
	sErrorDescription2 := 'Setup parameter and the power OFF';				
					
6520:					
					
	sErrorDescription1 := 'RS422 Parameter illgal.  Setup the parameter.';				
	sErrorDescription2 := 'Setup parameter and the power OFF';				
					
6530:					
					
	sErrorDescription1 := 'COMDEV parameter is illegal.  COMDEV parameter is illegal.';				
	sErrorDescription2 := 'Correct COMDEV parameter';				
					
6640:					
					
	sErrorDescription1 := 'Illegal param (special signal.  The parameter setting is illegal.';				
	sErrorDescription2 := 'Correct the parameter';				
					
6680:					
					
	sErrorDescription1 := ' Mismatch of Safety Input.  State of the redundant wiring do not match.(Safety Input).';				
	sErrorDescription2 := 'Please check the wiring or parameter';				
					
6681:					
					
	sErrorDescription1 := ' Mismatch of Safety Input1.  State of the redundant wiring do not match.(Safety Input 1).';				
	sErrorDescription2 := 'Please check the wiring or parameter';				
					
6682:					
					
	sErrorDescription1 := ' Mismatch of Safety Input2.  State of the redundant wiring do not match.(Safety Input 2).';				
	sErrorDescription2 := 'Please check the wiring or parameter';				
					
6683:					
					
	sErrorDescription1 := ' Mismatch of Safety Input3.  State of the redundant wiring do not match.(Safety Input 3).';				
	sErrorDescription2 := 'Please check the wiring or parameter';				
					
6690:					
					
	sErrorDescription1 := ' Safety Input Process error.  Abnormality of the Safety Input was detected.';				
	sErrorDescription2 := 'Turn the power OFF and ON once';				
					
7030:					
					
	sErrorDescription1 := 'System error (param size over.  Parameter file size over.';				
	sErrorDescription2 := 'Contact the maker';				
					
7050:					
					
	sErrorDescription1 := 'File is illegal.  The file is illegal.';				
	sErrorDescription2 := 'Do not use this file';				
					
7060:					
					
	sErrorDescription1 := 'System error (RAM area full).  System RAM area is full.';				
	sErrorDescription2 := 'Contact the maker';				
					
7100:					
					
	sErrorDescription1 := ' Robot arm serial number misma.  Robot arm that connection was replaced.';				
	sErrorDescription2 := 'Execute restoration of preventive maintenance data, or reset';				
					
7101:					
					
	sErrorDescription1 := ' Backup serial number mismatch.  Robot arm and backup data are the different serial number.';				
	sErrorDescription2 := 'Please use the backup data matching robot arm';				
					
7102:					
					
	sErrorDescription1 := ' Backup file version is differ.  Preventive maintenance function backup file version mismatch.';				
	sErrorDescription2 := 'Please select the backup file of the corresponding version';				
					
7300:					
					
	sErrorDescription1 := 'Loading the parameter file..  Turn the power OFF and ON once.';				
	sErrorDescription2 := 'Turn the power OFF and ON once';				
					
7600:					
					
	sErrorDescription1 := ' Illegal parameter (AXMENO).  The additional axis robot No. is incorrect.';				
	sErrorDescription2 := 'Correct parameter AXMENO,AXUNUM';				
					
7601:					
					
	sErrorDescription1 := ' Illegal parameter (AXJNO).  The additional axis No. is illegal.';				
	sErrorDescription2 := 'Correct parameter AXMENO';				
					
7602:					
					
	sErrorDescription1 := ' Duplicate parameter (AXJNO).  The additional axis No. has been used in duplicate.';				
	sErrorDescription2 := 'Correct parameter AXMENO';				
					
7603:					
					
	sErrorDescription1 := ' Illegal parameter (AXUNT).  The additional axis unit is incorrect.';				
	sErrorDescription2 := 'Correct parameter AXMUNT';				
					
7604:					
					
	sErrorDescription1 := ' Illegal parameter (AXACC).  The additional axis acceleration time is incorrect.';				
	sErrorDescription2 := 'Correct parameter AXACC';				
					
7605:					
					
	sErrorDescription1 := ' Illegal parameter (AXDCC).  The additional axis deceleration time is incorrect.';				
	sErrorDescription2 := 'Correct parameter AXDCC';				
					
7606:					
					
	sErrorDescription1 := ' Illegal parameter (AXGRTN).  The additional axis gear ratio denominator is incorrect.';				
	sErrorDescription2 := 'Correct parameter AXGRTN';				
					
7607:					
					
	sErrorDescription1 := ' Illegal parameter (AXGRTD).  The additional axis gear ratio numerator is incorrect.';				
	sErrorDescription2 := 'Correct parameter AXGRTD';				
					
7608:					
					
	sErrorDescription1 := ' Illegal parameter (AXMOTSET).  The additional axis motor setting validity flag is incorrect.';				
	sErrorDescription2 := 'Correct parameter AXMOTSET';				
					
7609:					
					
	sErrorDescription1 := ' Illegal parameter (AXMREV).  The additional axis motor rated speed is incorrect.';				
	sErrorDescription2 := 'Correct parameter AXMREV';				
					
7610:					
					
	sErrorDescription1 := ' Illegal parameter (AXJMX).  The additional axis motor limit speed is incorrect.';				
	sErrorDescription2 := 'Correct parameter AXJMX';				
					
7611:					
					
	sErrorDescription1 := ' Illegal parameter (AXENCR).  The additional axis No. of encoder pulses is incorrect.';				
	sErrorDescription2 := 'Correct parameter AXENCR';				
					
7612:					
					
	sErrorDescription1 := ' Illegal parameter (AXJOGTS).  The additional axis JOG time constant is incorrect.';				
	sErrorDescription2 := 'Correct parameter AXJOGTS';				
					
7613:					
					
	sErrorDescription1 := ' Turn the power OFF and ON onc.  Turn the power OFF and ON once.';				
	sErrorDescription2 := 'Turn the power OFF and ON once';				
					
7620:					
					
	sErrorDescription1 := ' Plural Add-Axis cards are set.  This card can install one.';				
	sErrorDescription2 := 'Reinstall one card';				
					
7650:					
					
	sErrorDescription1 := ' Number of force sensors is wr.  Two or more force sensors are set to one robot.';				
	sErrorDescription2 := 'Please confirm the setting of parameter AXJNO and AXMENO';				
					
7651:					
					
	sErrorDescription1 := ' I/F unit initialization error.  Initialization of the force control I/F unit failed.';				
	sErrorDescription2 := 'Please confirm the connection and the power supply of I/F unit';				
					
7652:					
					
	sErrorDescription1 := ' I/F unit revision is illegal.  It does not correspond to revision of this force sensor I/F unit.';				
	sErrorDescription2 := 'Please contact the maker';				
					
7660:					
					
	sErrorDescription1 := ' Force sensor error.  The data of force sensor that exceeded the limitation.';				
	sErrorDescription2 := 'Please confirm use and the state of force sensor';				
					
7700:					
					
	sErrorDescription1 := ' CC-Link card is illegal.  The master station is set.';				
	sErrorDescription2 := 'Please exchange the CC-Link card';				
					
7710:					
					
	sErrorDescription1 := ' Can not set the Master Station.  The master station is set..';				
	sErrorDescription2 := 'Set the station number except 0';				
					
7720:					
					
	sErrorDescription1 := ' Plural CC-Link cards are set.  CC-Link card can install one.';				
	sErrorDescription2 := 'Install only one CC-Link card';				
					
7760:					
					
	sErrorDescription1 := ' CC-Link initialization error.  Confirm the CC-Link error code.';				
	sErrorDescription2 := 'Confirm the CC-Link error code';				
					
7799:					
					
	sErrorDescription1 := ' CC-Link System error.  .';				
	sErrorDescription2 := '';				
					
7800:					
					
	sErrorDescription1 := ' Ethernet card initialization .  The Ethernet card is broken.';				
	sErrorDescription2 := 'Check the Ethernet board';				
					
7802:					
					
	sErrorDescription1 := ' Ethernet card is set in SLOT2.  Ethernet card is set in SLOT2 or 3.';				
	sErrorDescription2 := 'Install Ethernet card in SLOT1';				
					
7803:					
					
	sErrorDescription1 := ' Plural Ethernet cards are set.  Ethernet card can install one.';				
	sErrorDescription2 := 'Install the Ethernet card only in SLOT1';				
					
7810:					
					
	sErrorDescription1 := ' Ethernet parameter ERR.  Illegal parameter.';				
	sErrorDescription2 := 'Correct parameter';				
					
7820:					
					
	sErrorDescription1 := 'MXT/MXScommand timeout.  time over MXTTOUT parameter.';				
	sErrorDescription2 := 'Chech parameter MXTTOUT';				
					
7830:					
					
	sErrorDescription1 := 'Ethernet card is not installe.  Ethernet card is not installed, or command disable.';				
	sErrorDescription2 := 'Install Ethenet card';				
					
7840:					
					
	sErrorDescription1 := 'MXT/MXS command Illegal recei.  ・Illegal received data Illegal command position data (NAN/NUMBER) Different data type.';				
	sErrorDescription2 := 'Check MXT/MXS command and transmitted data Check transmitted command position data Check MXT/MXS command and transmitted data';				
					
7860:					
					
	sErrorDescription1 := ' SLMP error.  An error related to SLMP has occurred. .';				
	sErrorDescription2 := 'Please confirm the content by a detailed number of the error.';				
					
7861:					
					
	sErrorDescription1 := ' SLMP parameter error.  Illegal parameter. .';				
	sErrorDescription2 := 'Correct parameter. ';				
					
7870:					
					
	sErrorDescription1 := ' CC-Link IEF Basic Comm. Error.  Failure in the CC-Link IEF Commuication..';				
	sErrorDescription2 := 'Check the wiring and parameter setting on the master station.';				
					
7901:					
					
	sErrorDescription1 := ' OPTION1#1 Parameter illegal.  Setup the parameter.';				
	sErrorDescription2 := 'Setup patrameter and the power OFF';				
					
7902:					
					
	sErrorDescription1 := ' OPTION1#2 Parameter illegal.  Setup the parameter.';				
	sErrorDescription2 := 'Setup patrameter and the power OFF';				
					
7903:					
					
	sErrorDescription1 := ' OPTION1#3 Parameter illegal.  Setup the parameter.';				
	sErrorDescription2 := 'Setup patrameter and the power OFF';				
					
7911:					
					
	sErrorDescription1 := ' OPTION2#1 Parameter illegal.  Setup the parameter.';				
	sErrorDescription2 := 'Setup patrameter and the power OFF';				
					
7912:					
					
	sErrorDescription1 := ' OPTION2#2 Parameter illegal.  Setup the parameter.';				
	sErrorDescription2 := 'Setup patrameter and the power OFF';				
					
7913:					
					
	sErrorDescription1 := ' OPTION2#3 Parameter illegal.  Setup the parameter.';				
	sErrorDescription2 := 'Setup patrameter and the power OFF';				
					
7920:					
					
	sErrorDescription1 := ' Three EX-SIO I/F are installe.  Reinstall one or two cards to SLOT1 or 2.';				
	sErrorDescription2 := 'Remove the Expansion Serial card in SLOT3';				
					
7930:					
					
	sErrorDescription1 := ' EX-SIO card is set in SLOT3.  EX-SIO card is set in SLOT3.';				
	sErrorDescription2 := 'Remove the Expansion Serial card in SLOT 3';				
					
7990:					
					
	sErrorDescription1 := ' OptionCard illegal insert.  Check SLOT number.';				
	sErrorDescription2 := 'Power off, change the SLOT number';				
					
8000:					
					
	sErrorDescription1 := ' .  .';				
	sErrorDescription2 := '';				
					
8001:					
					
	sErrorDescription1 := ' .  .';				
	sErrorDescription2 := '';				
					
8002:					
					
	sErrorDescription1 := ' .  .';				
	sErrorDescription2 := '';				
					
8003:					
					
	sErrorDescription1 := ' .  .';				
	sErrorDescription2 := '';				
					
8004:					
					
	sErrorDescription1 := ' .  .';				
	sErrorDescription2 := '';				
					
8005:					
					
	sErrorDescription1 := ' .  .';				
	sErrorDescription2 := '';				
					
8010:					
					
	sErrorDescription1 := ' .  .';				
	sErrorDescription2 := '';				
					
8011:					
					
	sErrorDescription1 := ' .  .';				
	sErrorDescription2 := '';				
					
8012:					
					
	sErrorDescription1 := ' .  .';				
	sErrorDescription2 := '';				
					
8013:					
					
	sErrorDescription1 := ' .  .';				
	sErrorDescription2 := '';				
					
8014:					
					
	sErrorDescription1 := ' .  .';				
	sErrorDescription2 := '';				
					
8015:					
					
	sErrorDescription1 := ' Plural Vision cards are insta.  Vision card can be installed one.';				
	sErrorDescription2 := 'Reinstall one card';				
					
8016:					
					
	sErrorDescription1 := ' .  .';				
	sErrorDescription2 := '';				
					
8020:					
					
	sErrorDescription1 := ' .  .';				
	sErrorDescription2 := '';				
					
8021:					
					
	sErrorDescription1 := ' .  .';				
	sErrorDescription2 := '';				
					
8022:					
					
	sErrorDescription1 := ' .  .';				
	sErrorDescription2 := '';				
					
8023:					
					
	sErrorDescription1 := ' .  .';				
	sErrorDescription2 := '';				
					
8024:					
					
	sErrorDescription1 := ' .  .';				
	sErrorDescription2 := '';				
					
8025:					
					
	sErrorDescription1 := ' .  .';				
	sErrorDescription2 := '';				
					
8026:					
					
	sErrorDescription1 := ' .  .';				
	sErrorDescription2 := '';				
					
8027:					
					
	sErrorDescription1 := ' .  .';				
	sErrorDescription2 := '';				
					
8028:					
					
	sErrorDescription1 := ' .  .';				
	sErrorDescription2 := '';				
					
8029:					
					
	sErrorDescription1 := ' .  .';				
	sErrorDescription2 := '';				
					
8030:					
					
	sErrorDescription1 := ' .  .';				
	sErrorDescription2 := '';				
					
8031:					
					
	sErrorDescription1 := ' .  .';				
	sErrorDescription2 := '';				
					
8032:					
					
	sErrorDescription1 := ' .  .';				
	sErrorDescription2 := '';				
					
8033:					
					
	sErrorDescription1 := ' .  .';				
	sErrorDescription2 := '';				
					
8034:					
					
	sErrorDescription1 := ' .  .';				
	sErrorDescription2 := '';				
					
8035:					
					
	sErrorDescription1 := ' .  .';				
	sErrorDescription2 := '';				
					
8036:					
					
	sErrorDescription1 := ' .  .';				
	sErrorDescription2 := '';				
					
8037:					
					
	sErrorDescription1 := ' .  .';				
	sErrorDescription2 := '';				
					
8038:					
					
	sErrorDescription1 := ' .  .';				
	sErrorDescription2 := '';				
					
8039:					
					
	sErrorDescription1 := ' .  .';				
	sErrorDescription2 := '';				
					
8040:					
					
	sErrorDescription1 := ' .  .';				
	sErrorDescription2 := '';				
					
8130:					
					
	sErrorDescription1 := ' Multi-Hand Comm.error(RemoteI.  Communication line is illegal.';				
	sErrorDescription2 := 'Check the cable or power supply';				
					
8140:					
					
	sErrorDescription1 := ' Electric hand1 Comm.error(RIO.  Communication line is illegal.';				
	sErrorDescription2 := 'Check the cable or power supply';				
					
8150:					
					
	sErrorDescription1 := ' Electric hand2 Comm.error(RIO.  Communication line is illegal.';				
	sErrorDescription2 := 'Check the cable or power supply';				
					
8160:					
					
	sErrorDescription1 := ' Electric hand3 Comm.error(RIO.  Communication line is illegal.';				
	sErrorDescription2 := 'Check the cable or power supply';				
					
8201:					
					
	sErrorDescription1 := ' Illegal param (TPTMMG).  TPTMMG param is illegal.';				
	sErrorDescription2 := 'Correct TPTMMG parameter';				
					
8202:					
					
	sErrorDescription1 := ' Illegal param (TPERRNO).  TPERRNO param is illegal.';				
	sErrorDescription2 := 'Correct TPERRNO parameter';				
					
8203:					
					
	sErrorDescription1 := ' Illegal param (TPSIGNO).  TPSIGNO param is illegal.';				
	sErrorDescription2 := 'Correct TPSIGNO parameter';				
					
8204:					
					
	sErrorDescription1 := ' Illegal param (TRAP).  TRAP param is illegal.';				
	sErrorDescription2 := 'Correct TRAP parameter';				
					
8206:					
					
	sErrorDescription1 := ' failed in initialization (tra.  Turn the power OFF and power ON once.';				
	sErrorDescription2 := 'Please check communication state, setting, and command argument';				
					
8207:					
					
	sErrorDescription1 := ' failed in writing the data(tr.  failed in writing the data .';				
	sErrorDescription2 := 'Please do the operation over again';				
					
8320:					
					
	sErrorDescription1 := 'System Error (GETPOS).  Internal data of GETPOS is illegal.';				
	sErrorDescription2 := 'Turn the power OFF and ON once';				
					
8400:					
					
	sErrorDescription1 := 'CTN data is illegal (PREC or .  CTN data is illegal. It changed to PREC OFF and M_LDM=0..';				
	sErrorDescription2 := 'Try to set be a PREC mode and M_LDM again.';				
					
8410:					
					
	sErrorDescription1 := ' DEVICENET card failure.  Abnormality of the DEVICENET card is detected.';				
	sErrorDescription2 := 'Please exchange the DEVICENET card';				
					
8420:					
					
	sErrorDescription1 := ' DEVICENET Mode switch is outs.  The mode switch is outside.';				
	sErrorDescription2 := 'Please correct the mode switch';				
					
8421:					
					
	sErrorDescription1 := ' DEVICENET Unit number switch .  The unit number switch is outside.';				
	sErrorDescription2 := 'Please correct the unit number switch';				
					
8450:					
					
	sErrorDescription1 := ' DEVICENET Install more than o.  Only one TZ571 card can be installed.';				
	sErrorDescription2 := 'Please install only one TZ571 card';				
					
8451:					
					
	sErrorDescription1 := ' DEVICENET Set other fieldbus.  Only one. fieldbus card can be installed.';				
	sErrorDescription2 := 'Only one fieldbus card is installed';				
					
8470:					
					
	sErrorDescription1 := ' DEVICENET Param load write er.  Parameter can not be load and written.';				
	sErrorDescription2 := 'Turn the power OFF and ON once';				
					
8471:					
					
	sErrorDescription1 := ' DEVICENET Send byte is outsid.  Send byte number setting of is out of range.';				
	sErrorDescription2 := 'Please correct the send byte number setting';				
					
8472:					
					
	sErrorDescription1 := ' DEVICENET Receive byte outsid.  Receive byte number setting is outside.';				
	sErrorDescription2 := 'Please correct the ｒeceive byte number setting';				
					
8473:					
					
	sErrorDescription1 := ' DEVICENET Send-receive are 0.  Both receive and send byte number setting are 0.';				
	sErrorDescription2 := 'Please change receive or send byte number setting';				
					
8491:					
					
	sErrorDescription1 := ' DEVICENET Comm-test unit numb.  Unit numbers overlap is detected by communication test.';				
	sErrorDescription2 := 'Please confirm the other units number';				
					
8492:					
					
	sErrorDescription1 := ' DEVICENET Comm-test busoff.  Busoff is detected by communication test.';				
	sErrorDescription2 := 'Please confirm communication speed,cable,terminator';				
					
8493:					
					
	sErrorDescription1 := ' DEVICENET Comm-test net power.  Network power off is detected by communication test.';				
	sErrorDescription2 := 'Please turn on network power';				
					
8494:					
					
	sErrorDescription1 := ' DEVICENET Comm-test send-rece.  Data can not send and recive normal by communication test.';				
	sErrorDescription2 := 'Please confirm connection, comm speed, cable and terminator';				
					
8500:					
					
	sErrorDescription1 := ' PROFIBUS Initial error.  Hardware is abnormal..';				
	sErrorDescription2 := 'Please exchange the PROFIBUS TZ577 card.';				
					
8501:					
					
	sErrorDescription1 := ' PROFIBUS watch dog timer erro.  Hardware is abnormal..';				
	sErrorDescription2 := 'Please exchange the PROFIBUS TZ577 card.';				
					
8502:					
					
	sErrorDescription1 := ' Plural PROFIBUS cards are set.  PROFIBUS card can be installed one..';				
	sErrorDescription2 := 'Install only one PROFIBUS card.';				
					
8503:					
					
	sErrorDescription1 := ' PROFIBUS/CC-Link cards are se.  PROFIBUS card can be installed one..';				
	sErrorDescription2 := 'Install only either of of one PROFIBUS or one CC-Link card.';				
					
8504:					
					
	sErrorDescription1 := ' PROFIBUS self-check error.  Hardware is abnormal..';				
	sErrorDescription2 := 'Please exchange the PROFIBUS TZ577 card.';				
					
8505:					
					
	sErrorDescription1 := ' Illegal param (PBMODE).  PBMODE param is illegal.';				
	sErrorDescription2 := 'Correct PBMODE parameter (0 or 2)';				
					
8506:					
					
	sErrorDescription1 := ' Exchange number cannot be set.  Turn the power off and ON once.';				
	sErrorDescription2 := 'The card might be broken. Please repair it.';				
					
8507:					
					
	sErrorDescription1 := ' Illegal param (PBMC).  PBMC param is illegal.';				
	sErrorDescription2 := 'Correct PBMC parameter (1:Class / 2:Class2)';				
					
8510:					
					
	sErrorDescription1 := ' PROFIBUS exchange NO.is wrong.  The exchange number is outside the range..';				
	sErrorDescription2 := 'Please set PBNUM Parameter within the range of -1 to 125.';				
					
8520:					
					
	sErrorDescription1 := ' PROFIBUS St.number write erro.  The exchange Station Number is protected..';				
	sErrorDescription2 := 'Set -1 to the exchange Station Number.';				
					
8530:					
					
	sErrorDescription1 := ' PROFIBUS St.number write erro.  Exchange St.number is continuously rewritten 60 times or more..';				
	sErrorDescription2 := 'Please exchange the PROFIBUS TZ577 card.';				
					
8540:					
					
	sErrorDescription1 := ' PROFIBUS flash ROM access err.  Hardware is abnormal..';				
	sErrorDescription2 := 'Please exchange the PROFIBUS TZ577 card.';				
					
8550:					
					
	sErrorDescription1 := ' PROFIBUS master bureaus para.  The parameter settting in the master is illegal.';				
	sErrorDescription2 := 'Please confirm the slave parameter of the master bureau';				
					
8560:					
					
	sErrorDescription1 := ' PROFIBUS communication chip E.  Hardware is broken.';				
	sErrorDescription2 := 'Please exchange the PROFIBUS TZ577 card.';				
					
8570:					
					
	sErrorDescription1 := ' PROFIBUS communication Time-o.  The time-out was generated by the communication with the master..';				
	sErrorDescription2 := 'Check the masters state, the cable and lengthen WDT.';				
					
8580:					
					
	sErrorDescription1 := ' PROFIBUS I/O composition erro.  The data module is not a word type..';				
	sErrorDescription2 := 'Confirm the slave parameter. (Refer to masters manual)';				
					
8740:					
					
	sErrorDescription1 := ' CR800 init communication erro.  Initial communication with the CR800 was not possible.';				
	sErrorDescription2 := 'Check the communication cable connection';				
					
8741:					
					
	sErrorDescription1 := ' CPU unit init communication e.  Initial communication with the CPU unit was not possible.';				
	sErrorDescription2 := 'Check the communication cable connection';				
					
8751:					
					
	sErrorDescription1 := ' CR800 communication error.  Communication from the CR800 was cut off.';				
	sErrorDescription2 := 'Check the communication cable connection';				
					
8752:					
					
	sErrorDescription1 := ' CPU unit communication error.  Communication from the CPU unit was cut off.';				
	sErrorDescription2 := 'Check the communication cable connection';				
					
8760:					
					
	sErrorDescription1 := ' PLC CPU parameters are not se.  Fixed Scan Communication Area is not set in the PLC CPU.';				
	sErrorDescription2 := 'Please set the Fixed Scan Communication Area in the PLC CPU';				
					
8761:					
					
	sErrorDescription1 := ' CPU number setting is illegal.  The setting of CPU number is different.';				
	sErrorDescription2 := 'Please check PLC multi CPU setting and QMLTCPUN parameter';				
					
8762:					
					
	sErrorDescription1 := ' Multi-CPU parameter is illega.  There is a mistake in setting of a multi-CPU parameter.';				
	sErrorDescription2 := 'Please confirm the set value and change it to the right value';				
					
8770:					
					
	sErrorDescription1 := ' CR800 communication error.  Communication error was detected from CR800.';				
	sErrorDescription2 := 'Check the communication cable connection';				
					
8780:					
					
	sErrorDescription1 := ' CPU unit communication error.  Communication error was detected from the CPU unit.';				
	sErrorDescription2 := 'Check the communication cable connection';				
					
8790:					
					
	sErrorDescription1 := ' CR800 error reset error.  Can not reset CR800 error.';				
	sErrorDescription2 := 'Check the communication cable connection';				
					
8800:					
					
	sErrorDescription1 := 'ASIC communication error.  ・Error occurred by the data reception from the servo CRC error in the receive data from the servo Abnormal data was received from the servo Abnormal data was received from the servo Connection is defective of the com. cable Empty data was.';				
	sErrorDescription2 := 'Check the communication cable connection';				
					
8810:					
					
	sErrorDescription1 := 'Communication error.  ・Error occurred by the data transmission to the servo ID of the com. data with the servo is not corresponding.';				
	sErrorDescription2 := 'Check the communication cable connection';				
					
8820:					
					
	sErrorDescription1 := 'Communication timeout.  The communication with the servo became a timeout.';				
	sErrorDescription2 := 'Turn the power OFF and ON once';				
					
8830:					
					
	sErrorDescription1 := 'Amplifier unconnection.  ・The servo amplifier cannot be detected The axis setting is not correct Uncorrespondence amplifier is connected The communication protocol which does not correspond Uncorrespondence motor is connected A set value of the servo parameter is.';			
	sErrorDescription2 := '・Check the cable connection and the power supply of amp. Check the servo axis settings (parameters, rotary switches) Remove the uncorrespondence amplifier Remove the uncorrespondence motor';				
					
8841:					
					
	sErrorDescription1 := ' Illegal number of add. axis c.  Two or more addition axis I/F cards are installed.';				
	sErrorDescription2 := 'Adjust addition axis I/F card to one piece';				
					
8860:					
					
	sErrorDescription1 := ' Illegal protocol specificatio.  The specification of the servo protocol is wrong.';				
	sErrorDescription2 := 'Check the parameter SVNETSTD';				
					
8870:					
					
	sErrorDescription1 := 'Transient processing error.  Illegal demand data was transmitted.';				
	sErrorDescription2 := 'Check the demand data';				
					
8920:					
					
	sErrorDescription1 := ' Error of sensor I/F unit.  The error occurred by sensor I/F unit.';				
	sErrorDescription2 := 'Please refer to the manual of sensor I/F unit';				
					
9000:					
					
	sErrorDescription1 := 'Opening gripper Error';				
	sErrorDescription2 := 'Check Gripper';				
					
9001:					
					
	sErrorDescription1 := 'Closing gripper Error';				
	sErrorDescription2 := 'Check Gripper';				
					
9002:					
					
	sErrorDescription1 := 'User High level error.  Illegal demand data was transmitted.';				
	sErrorDescription2 := 'Check program';				
					
9003:					
					
	sErrorDescription1 := 'User High level error.  Illegal demand data was transmitted.';				
	sErrorDescription2 := 'Check program';				
					
9004:					
					
	sErrorDescription1 := 'User High level error.  Illegal demand data was transmitted.';				
	sErrorDescription2 := 'Check program';				
					
9005:					
					
	sErrorDescription1 := 'User High level error.  Illegal demand data was transmitted.';				
	sErrorDescription2 := 'Check program';				
					
9006:					
					
	sErrorDescription1 := 'User High level error.  Illegal demand data was transmitted.';				
	sErrorDescription2 := 'Check program';				
					
9007:					
					
	sErrorDescription1 := 'User High level error.  Illegal demand data was transmitted.';				
	sErrorDescription2 := 'Check program';				
					
9008:					
					
	sErrorDescription1 := 'User High level error.  Illegal demand data was transmitted.';				
	sErrorDescription2 := 'Check program';				
					
9009:					
					
	sErrorDescription1 := 'User High level error.  Illegal demand data was transmitted.';				
	sErrorDescription2 := 'Check program';				
					
9010:					
					
	sErrorDescription1 := 'User High level error.  Illegal demand data was transmitted.';				
	sErrorDescription2 := 'Check program';				
					
9011:					
					
	sErrorDescription1 := 'User High level error.  Illegal demand data was transmitted.';				
	sErrorDescription2 := 'Check program';				
					
9012:					
					
	sErrorDescription1 := 'User High level error.  Illegal demand data was transmitted.';				
	sErrorDescription2 := 'Check program';				
					
9013:					
					
	sErrorDescription1 := 'User High level error.  Illegal demand data was transmitted.';				
	sErrorDescription2 := 'Check program';				
					
9014:					
					
	sErrorDescription1 := 'User High level error.  Illegal demand data was transmitted.';				
	sErrorDescription2 := 'Check program';				
					
9015:					
					
	sErrorDescription1 := 'User High level error.  Illegal demand data was transmitted.';				
	sErrorDescription2 := 'Check program';				
					
9016:					
					
	sErrorDescription1 := 'User High level error.  Illegal demand data was transmitted.';				
	sErrorDescription2 := 'Check program';				
					
9017:					
					
	sErrorDescription1 := 'User High level error.  Illegal demand data was transmitted.';				
	sErrorDescription2 := 'Check program';				
					
9018:					
					
	sErrorDescription1 := 'User High level error.  Illegal demand data was transmitted.';				
	sErrorDescription2 := 'Check program';				
					
9019:					
					
	sErrorDescription1 := 'User High level error.  Illegal demand data was transmitted.';				
	sErrorDescription2 := 'Check program';				
					
9020:					
					
	sErrorDescription1 := 'User High level error.  Illegal demand data was transmitted.';				
	sErrorDescription2 := 'Check program';				
					
9021:					
					
	sErrorDescription1 := 'User High level error.  Illegal demand data was transmitted.';				
	sErrorDescription2 := 'Check program';				
					
9022:					
					
	sErrorDescription1 := 'User High level error.  Illegal demand data was transmitted.';				
	sErrorDescription2 := 'Check program';				
					
9023:					
					
	sErrorDescription1 := 'User High level error.  Illegal demand data was transmitted.';				
	sErrorDescription2 := 'Check program';				
					
9024:					
					
	sErrorDescription1 := 'User High level error.  Illegal demand data was transmitted.';				
	sErrorDescription2 := 'Check program';				
					
9025:					
					
	sErrorDescription1 := 'User High level error.  Illegal demand data was transmitted.';				
	sErrorDescription2 := 'Check program';				
					
9026:					
					
	sErrorDescription1 := 'User High level error.  Illegal demand data was transmitted.';				
	sErrorDescription2 := 'Check program';				
					
9027:					
					
	sErrorDescription1 := 'User High level error.  Illegal demand data was transmitted.';				
	sErrorDescription2 := 'Check program';				
					
9028:					
					
	sErrorDescription1 := 'User High level error.  Illegal demand data was transmitted.';				
	sErrorDescription2 := 'Check program';				
					
9029:					
					
	sErrorDescription1 := 'User High level error.  Illegal demand data was transmitted.';				
	sErrorDescription2 := 'Check program';				
					
9030:					
					
	sErrorDescription1 := 'User High level error.  Illegal demand data was transmitted.';				
	sErrorDescription2 := 'Check program';				
					
9031:					
					
	sErrorDescription1 := 'User High level error.  Illegal demand data was transmitted.';				
	sErrorDescription2 := 'Check program';				
					
9032:					
					
	sErrorDescription1 := 'User High level error.  Illegal demand data was transmitted.';				
	sErrorDescription2 := 'Check program';				
					
9033:					
					
	sErrorDescription1 := 'User High level error.  Illegal demand data was transmitted.';				
	sErrorDescription2 := 'Check program';				
					
9034:					
					
	sErrorDescription1 := 'User High level error.  Illegal demand data was transmitted.';				
	sErrorDescription2 := 'Check program';				
					
9035:					
					
	sErrorDescription1 := 'User High level error.  Illegal demand data was transmitted.';				
	sErrorDescription2 := 'Check program';				
					
9036:					
					
	sErrorDescription1 := 'User High level error.  Illegal demand data was transmitted.';				
	sErrorDescription2 := 'Check program';				
					
9037:					
					
	sErrorDescription1 := 'User High level error.  Illegal demand data was transmitted.';				
	sErrorDescription2 := 'Check program';				
					
9038:					
					
	sErrorDescription1 := 'User High level error.  Illegal demand data was transmitted.';				
	sErrorDescription2 := 'Check program';				
					
9039:					
					
	sErrorDescription1 := 'User High level error.  Illegal demand data was transmitted.';				
	sErrorDescription2 := 'Check program';				
					
9040:					
					
	sErrorDescription1 := 'User High level error.  Illegal demand data was transmitted.';				
	sErrorDescription2 := 'Check program';				
					
9041:					
					
	sErrorDescription1 := 'User High level error.  Illegal demand data was transmitted.';				
	sErrorDescription2 := 'Check program';				
					
9042:					
					
	sErrorDescription1 := 'User High level error.  Illegal demand data was transmitted.';				
	sErrorDescription2 := 'Check program';				
					
9043:					
					
	sErrorDescription1 := 'User High level error.  Illegal demand data was transmitted.';				
	sErrorDescription2 := 'Check program';				
					
9044:					
					
	sErrorDescription1 := 'User High level error.  Illegal demand data was transmitted.';				
	sErrorDescription2 := 'Check program';				
					
9045:					
					
	sErrorDescription1 := 'User High level error.  Illegal demand data was transmitted.';				
	sErrorDescription2 := 'Check program';				
					
9046:					
					
	sErrorDescription1 := 'User High level error.  Illegal demand data was transmitted.';				
	sErrorDescription2 := 'Check program';				
					
9047:					
					
	sErrorDescription1 := 'User High level error.  Illegal demand data was transmitted.';				
	sErrorDescription2 := 'Check program';				
					
9048:					
					
	sErrorDescription1 := 'User High level error.  Illegal demand data was transmitted.';				
	sErrorDescription2 := 'Check program';				
					
9049:					
					
	sErrorDescription1 := 'User High level error.  Illegal demand data was transmitted.';				
	sErrorDescription2 := 'Check program';				
					
9050:					
					
	sErrorDescription1 := 'User High level error.  Illegal demand data was transmitted.';				
	sErrorDescription2 := 'Check program';				
					
9051:					
					
	sErrorDescription1 := 'User High level error.  Illegal demand data was transmitted.';				
	sErrorDescription2 := 'Check program';				
					
9052:					
					
	sErrorDescription1 := 'User High level error.  Illegal demand data was transmitted.';				
	sErrorDescription2 := 'Check program';				
					
9053:					
					
	sErrorDescription1 := 'User High level error.  Illegal demand data was transmitted.';				
	sErrorDescription2 := 'Check program';				
					
9054:					
					
	sErrorDescription1 := 'User High level error.  Illegal demand data was transmitted.';				
	sErrorDescription2 := 'Check program';				
					
9055:					
					
	sErrorDescription1 := 'User High level error.  Illegal demand data was transmitted.';				
	sErrorDescription2 := 'Check program';				
					
9056:					
					
	sErrorDescription1 := 'User High level error.  Illegal demand data was transmitted.';				
	sErrorDescription2 := 'Check program';				
					
9057:					
					
	sErrorDescription1 := 'User High level error.  Illegal demand data was transmitted.';				
	sErrorDescription2 := 'Check program';				
					
9058:					
					
	sErrorDescription1 := 'User High level error.  Illegal demand data was transmitted.';				
	sErrorDescription2 := 'Check program';				
					
9059:					
					
	sErrorDescription1 := 'User High level error.  Illegal demand data was transmitted.';				
	sErrorDescription2 := 'Check program';				
					
9060:					
					
	sErrorDescription1 := 'User High level error.  Illegal demand data was transmitted.';				
	sErrorDescription2 := 'Check program';				
					
9061:					
					
	sErrorDescription1 := 'User High level error.  Illegal demand data was transmitted.';				
	sErrorDescription2 := 'Check program';				
					
9062:					
					
	sErrorDescription1 := 'User High level error.  Illegal demand data was transmitted.';				
	sErrorDescription2 := 'Check program';				
					
9063:					
					
	sErrorDescription1 := 'User High level error.  Illegal demand data was transmitted.';				
	sErrorDescription2 := 'Check program';				
					
9064:					
					
	sErrorDescription1 := 'User High level error.  Illegal demand data was transmitted.';				
	sErrorDescription2 := 'Check program';				
					
9065:					
					
	sErrorDescription1 := 'User High level error.  Illegal demand data was transmitted.';				
	sErrorDescription2 := 'Check program';				
					
9066:					
					
	sErrorDescription1 := 'User High level error.  Illegal demand data was transmitted.';				
	sErrorDescription2 := 'Check program';				
					
9067:					
					
	sErrorDescription1 := 'User High level error.  Illegal demand data was transmitted.';				
	sErrorDescription2 := 'Check program';				
					
9068:					
					
	sErrorDescription1 := 'User High level error.  Illegal demand data was transmitted.';				
	sErrorDescription2 := 'Check program';				
					
9069:					
					
